// TIA Portal V17 export
// export: Created 2022-07-20T06:59:40.0910182Z, ExportSetting WithDefaults, DisplayName Totally Integrated Automation Portal, DisplayVersion V17, DisplayName TIA Portal Openness, DisplayVersion V17, DisplayName TIA Portal Version Control Interface, DisplayVersion V17, DisplayName SINAMICS Startdrive Advanced, DisplayVersion V17, DisplayName SINAMICS Startdrive G130, G150, S120, S150, SINAMICS MV, S210, DisplayVersion V17, DisplayName SINAMICS Startdrive G110M, G120, G120C, G120D, G120P, G115D, DisplayVersion V17, DisplayName STEP 7 Professional, DisplayVersion V17, DisplayName STEP 7 Safety, DisplayVersion V17, DisplayName WinCC Advanced, DisplayVersion V17
FUNCTION "FC10019_RealToString" : String   // FC10019, LAD
{ S7_Optimized_Access := 'TRUE' }
VERSION : 0.1
// stored: AutoNumber false, IsIECCheckEnabled false, SetENOAutomatically false, UDAEnableTagReadback false
   VAR_INPUT
      Real_In : Real;
   END_VAR
   VAR_TEMP
      String_Temp : String;
   END_VAR
BEGIN

REGION Network 1 (SCL): Real To String Management
   IF #Real_In <> 0.0 THEN
       #String_Temp := DINT_TO_STRING(REAL_TO_DINT(TRUNC_REAL(#Real_In * 10000)));
       #FC10019_RealToString := INSERT(IN1 := #String_Temp, IN2 := '.', P := LEN(#String_Temp) - 4);
   ELSE
       #FC10019_RealToString := '0.0';
   END_IF;
END_REGION
END_FUNCTION
